// SIMATIC S7-200 project (STEP 7-Micro/WIN), CPU 224 REL 02.00

SYMBOL_TABLE 符号表
AO_B             AQW0     // 板链线变频器DC0-10V信号
AO_X             AQW2     // 悬挂线变频器DC0-10V信号
C_1              C1       // 板链线运行工位计数
C_2              C2       // 悬挂线运行工位计数
HC_0             HC0      // 板链线编码器脉冲检测高速计数器
HC_1             HC1      // 板链线编码器脉冲检测高速计数器
BMQ_B            I0.0     // 板链线编码器
SP_B             I0.1     // 板链线接近开关
SF1_B            I0.2     // 板链线单独启动
SS1_B            I0.3     // 板链线单独停止
SFA_B            I0.4     // 板链线速度微增
SFD_B            I0.5     // 板链线速度微减
BMQ_X            I0.6     // 悬挂线编码器
SP_X             I0.7     // 悬挂线接近开关
SF1_X            I1.0     // 悬挂线单独启动
SS1_X            I1.1     // 悬挂线单独停止
SFA_X            I1.2     // 悬挂线速度微增
SFD_X            I1.3     // 悬挂线速度微减
SF1              I1.4     // 同步连续运行启动
SS1              I1.5     // 同步连续运行停止
BPQ_B            I2.0     // 板链线变频器故障
BPQ_X            I2.1     // 悬挂线变频器故障
SS2              I2.2     // 同步节拍运行停止
SF2              I2.3     // 同步节拍运行启动
M1_0             M1.0     // 板链线单独连续运行
M1_1             M1.1     // 悬挂线单独连续运行
M1_2             M1.2     // 板链线、悬挂线同步节拍运行
M1_3             M1.3     // 板链线、悬挂线同步节拍运行上升沿微分
M1_4             M1.4     // 板链线、悬挂线同步节拍运行状态下板链线接近开关上升沿微分
M1_5             M1.5     // 板链线、悬挂线同步节拍运行状态之板链线运行
M2_4             M2.4     // 板链线、悬挂线同步节拍运行状态下悬挂线接近开关上升沿微分
M2_5             M2.5     // 板链线、悬挂线同步节拍运行状态之悬挂线运行
M2_7             M2.7     // 板链线、悬挂线同步连续运行
M3_0             M3.0     // 板链线变频器复位状态
M3_1             M3.1     // 悬挂线变频器复位状态
M3_4             M3.4     // 单独连续运行开环控制方式
M3_5             M3.5     // 计数器复位
M4_1             M4.1     // C1>C2的下降沿
M4_2             M4.2     // C1<C2的下降沿
HL1              Q0.0     // 同步运行指示
HL2              Q0.1     // 同步停止指示
HL_B             Q0.2     // 板链线单独运行指示
HL_X             Q0.3     // 悬挂线单独运行指示
FWD_B            Q0.4     // 板链线正转
BX1_B            Q0.5     // 板链线自由停止
RST_B            Q0.6     // 板链线变频器复位
FWD_X            Q0.7     // 悬挂线正转
BX1_X            Q1.0     // 悬挂线自由停止
RST_X            Q1.1     // 悬挂线变频器复位
HLA_B            Q2.0     // 板链线速度微增指示
HLD_B            Q2.1     // 板链线速度微减指示
HLA_X            Q2.2     // 悬挂线速度微增指示
HLD_X            Q2.3     // 悬挂线速度微减指示
SM0_0            SM0.0    // 该位始终为1
SM0_1            SM0.1    // 首次扫描时SM0.1=1
SMB_37           SMB37    // HSC0的控制字节
SMB_47           SMB47    // HSC1的控制字节
SMD_38           SMD38    // HSC0的初始值(双整数)
SMD_42           SMD42    // HSC0的预置值(双整数)
SMD_48           SMD48    // HSC1的初始值(双整数)
SMD_52           SMD52    // HSC1的预置值(双整数)
T_0              T0       // 用于检测板链线夹具比悬挂线吊篮早到达接近开关的时间的ms定时器
T_32             T32      // 线体速度计算ms定时器
T_37             T37      // 单独连续运行开环控制状态持续时间
T_40             T40      // 板链线变频器复位持续时间
T_41             T41      // 悬挂线变频器复位持续时间
T_64             T64      // 用于检测悬挂线吊篮比板链线夹具早到达接近开关的时间的ms定时器
T_97             T97      // 板链线频率微增、微减时钟
T_98             T98      // 悬挂线频率微增、微减时钟
T_101            T101     // 板链线、悬挂线同步节拍运行状态下装配（停止）时间
T_105            T105     // 板链线、悬挂线同步连续运行启动时间
T_255            T255     // C1=C2计时
VD_40            VD40     // 板链线设定速度(米/分钟,实数)
VD_60            VD60     // 板链线实际运行速度(米/分钟,实数)
VD_80            VD80     // 悬挂线设定速度(米/分钟,实数)
VD_100           VD100    // 悬挂线实际运行速度(米/分钟,实数)
VD_140           VD140    // 板链线主动链轮节圆周长(米,实数)
VD_160           VD160    // 悬挂线主动链轮节圆周长(米,实数)
VD_240           VD240    // 板链线夹具间距=悬挂线吊篮间距(米,实数)
VD_1800          VD1800   // 线体速度计算采样脉冲数(双整数)
VD_1804          VD1804   // 线体速度计算采样脉冲数(实数)
VD_1854          VD1854   // 检测指定数量脉冲所需要的时间(ms,双整数)
VD_2000          VD2000   // 板链线速度采样周期内的编码器脉冲数(个,双整数)
VD_2004          VD2004   // 板链线速度采样周期内的编码器脉冲数(个,实数)
VD_2008          VD2008   // 板链线编码器的分辨率(个脉冲/转,双整数)
VD_2012          VD2012   // 板链线编码器的分辨率(个脉冲/转,实数)
VD_2016          VD2016   // 线体速度计算采样周期(秒,双整数)
VD_2020          VD2020   // 线体速度计算采样周期(秒,实数)
VD_2024          VD2024   // 板链线速度计算中间值1(实数)
VD_2028          VD2028   // 板链线速度计算中间值2(实数)
VD_2032          VD2032   // 板链线速度计算中间值3(实数)
VD_2100          VD2100   // 检测指定数量脉冲所需要的时间(ms,双整数)
VD_2104          VD2104   // 检测指定数量脉冲所需要的时间(ms,实数)
VD_2108          VD2108   // 悬挂线编码器的分辨率(个脉冲/转,双整数)
VD_2112          VD2112   // 悬挂线编码器的分辨率(个脉冲/转,实数)
VD_2124          VD2124   // 悬挂线速度计算中间值1(实数)
VD_2128          VD2128   // 悬挂线速度计算中间值2(实数)
VD_2132          VD2132   // 悬挂线速度计算中间值3(实数)
VD_2204          VD2204   // 板链线夹具比悬挂线吊篮早到达接近开关的时间(ms,双整数)
VD_2208          VD2208   // 板链线夹具比悬挂线吊篮早到达接近开关的时间(ms,实数)
VD_2212          VD2212   // 速度偏差计算(板链线快)中间变量1
VD_2216          VD2216   // 速度偏差计算(板链线快)中间变量2
VD_2220          VD2220   // 速度偏差计算(板链线快)中间变量3
VD_2224          VD2224   // 速度偏差计算(板链线快)中间变量4
VD_2228          VD2228   // 速度偏差计算(板链线快)中间变量5
VD_2232          VD2232   // 板链线速度-悬挂线速度的值(正值)
VD_2304          VD2304   // 悬挂线吊篮比板链线夹具早到达接近开关的时间(ms,双整数)
VD_2308          VD2308   // 悬挂线吊篮比板链线夹具早到达接近开关的时间(ms,实数)
VD_2312          VD2312   // 速度偏差计算(悬挂线快)中间变量1
VD_2316          VD2316   // 速度偏差计算(悬挂线快)中间变量2
VD_2320          VD2320   // 速度偏差计算(悬挂线快)中间变量3
VD_2324          VD2324   // 速度偏差计算(板链线快)中间变量4
VD_2328          VD2328   // 速度偏差计算(板链线快)中间变量5
VD_2332          VD2332   // 悬挂线速度的值-板链线速度(正值)
VD_2336          VD2336   // 板链线速度-悬挂线速度的值(负值)
VD_2400          VD2400   // 板链线实际运行速度------PID反馈信号处理中间变量1(实数)
VD_2404          VD2404   // 板链线实际运行速度------PID反馈信号处理中间变量2(双整数)
VD_2420          VD2420   // 板链线设定速度------PID设定信号处理结果(实数)
VD_2440          VD2440   // 悬挂线实际运行速度------PID反馈信号处理中间变量1(实数)
VD_2444          VD2444   // 悬挂线实际运行速度------PID反馈信号处理中间变量2(双整数)
VD_2460          VD2460   // 悬挂线单独连续运行、同步节拍运行设定速度------PID设定信号处理中间变量1(实数)
VD_2500          VD2500   // 板链线速度-悬挂线速度的值(实数)
VD_2504          VD2504   // 悬挂线同步连续运行设定速度------PID设定信号处理中间变量2(实数)
VD_2508          VD2508   // 悬挂线同步连续运行设定速度------PID设定信号处理结果
VD_2600          VD2600   // 板链线单独连续开环运行设定速度换算中间变量1(实数)
VD_2604          VD2604   // 板链线单独连续开环运行设定速度换算中间变量2(实数)
VD_2608          VD2608   // 板链线单独连续开环运行设定速度换算中间变量3(双整数)
VD_2700          VD2700   // 悬挂线单独连续开环运行设定速度换算中间变量1(实数)
VD_2704          VD2704   // 悬挂线单独连续开环运行设定速度换算中间变量2(实数)
VD_2708          VD2708   // 悬挂线单独连续开环运行设定速度换算中间变量3(双整数)
VW_122           VW122    // 单独连续运行控制方式（1为开环控制，否则为PID控制）
VW_182           VW182    // 板链线编码器的分辨率(个脉冲/转,整数)
VW_202           VW202    // 悬挂线编码器的分辨率(个脉冲/转,整数)
VW_222           VW222    // 线体速度计算采样脉冲数(整数)
VW_226           VW226    // 线体速度计算采样周期(毫秒,整数)
VW_262           VW262    // PLC复位信号
VW_282           VW282    // 同步节拍运行时间(秒,整数)
VW_1850          VW1850   // 检测指定数量脉冲所需要的时间(ms,整数)
VW_1900          VW1900   // 同步节拍运行时间(百毫秒,整数)
VW_2200          VW2200   // 板链线夹具比悬挂线吊篮早到达接近开关的时间(ms,整数)
VW_2300          VW2300   // 悬挂线吊篮比板链线夹具早到达接近开关的时间(ms,整数)
VW_2408          VW2408   // 板链线实际运行速度------PID反馈信号处理结果(整数)
VW_2448          VW2448   // 悬挂线实际运行速度------PID反馈信号处理结果(整数)
VW_2612          VW2612   // 板链线单独连续开环运行设定速度换算中间变量4(整数)
VW_2712          VW2712   // 悬挂线单独连续开环运行设定速度换算中间变量4(整数)
END_SYMBOL_TABLE

ORGANIZATION_BLOCK 同步控制系统:OB1
TITLE=概要
// 这个PLC程序是给新大洲本田摩托车有限公司上海分公司设计的整车装配板链线和零件输送悬挂线同步控制系统改造工程。
// 项目实现摩托车装配线的自动化生产，通过同步控制板链线和悬挂线的运行来匹配装配节拍。
// 系统支持板链线单独连续运行、悬挂线单独连续运行、同步节拍运行和同步连续运行四种模式，且运行模式互斥。设备要求包含板链线输送设备、悬挂线输送设备、接近开关、高速计数器和变频器。
// 系统启动时，首次扫描标志在 PLC 上电后的第一个周期置 1，触发初始化逻辑。
// 程序支持四种运行模式：板链线单独连续运行、悬挂线单独连续运行、同步节拍运行和同步连续运行，这些模式通过按钮触发，但板链线单独连续运行标志、悬挂线单独连续运行标志、同步节拍运行标志和同步连续运行标志在任意时刻只能有一个为真，其他必须为假，确保车间内不会出现模式冲突导致的生产中断。
BEGIN
Network 1 // 系统初始化
// PLC上电运行的第一个扫描周期执行一次初始化子程序SBR_0，用于程序运行的初始设置
LD     SM0_1:SM0.1
CALL   线体实际速度计算初始化:SBR0
Network 2
// PLC上电运行的第一个扫描周期定义系统参数
LD     SM0_1:SM0.1
MOVR   1.37288, VD_140:VD140
MOVR   0.524271, VD_160:VD160
MOVR   2.4, VD_240:VD240
MOVW   360, VW_182:VW182
MOVW   360, VW_202:VW202
MOVW   50, VW_222:VW222
Network 3 // 板链线单独连续运行
// 板链线单独连续启动、停止、运行指示
LD     SF1_B:I0.2
O      M1_0:M1.0
AN     SS1_B:I0.3
AN     BPQ_B:I2.0
AN     M1_2:M1.2
AN     M2_7:M2.7
=      M1_0:M1.0
=      HL_B:Q0.2
Network 4 // 悬挂线单独连续运行
// 悬挂线单独连续启动、停止、运行指示
LD     SF1_X:I1.0
O      M1_1:M1.1
AN     SS1_X:I1.1
AN     BPQ_X:I2.1
AN     M1_2:M1.2
AN     M2_7:M2.7
=      M1_1:M1.1
=      HL_X:Q0.3
Network 5 // 板链线、悬挂线同步节拍运行
// 板链线、悬挂线同步节拍启动、停止
LD     SF2:I2.3
O      M1_2:M1.2
AN     SS2:I2.2
AN     BPQ_B:I2.0
AN     BPQ_X:I2.1
AN     M1_0:M1.0
AN     M2_7:M2.7
=      M1_2:M1.2
Network 6 // 板链线、悬挂线节拍同步运行装配（停止）时间单位转换
// 把节拍同步运行装配（停止）时间由秒转换为百毫秒
LD     M1_2:M1.2
MOVW   VW_282:VW282, VW_1900:VW1900
*I     +10, VW_1900:VW1900
Network 7 // 板链线、悬挂线同步节拍运行上升沿微分
LD     M1_2:M1.2
EU
=      M1_3:M1.3
Network 8 // 板链线、悬挂线同步节拍运行状态下板链线接近开关上升沿微分
LD     M1_2:M1.2
A      SP_B:I0.1
EU
=      M1_4:M1.4
Network 9 // 板链线、悬挂线同步节拍运行状态之板链线运行
LD     M1_3:M1.3
O      M1_5:M1.5
O      T_101:T101
A      M1_2:M1.2
AN     M1_4:M1.4
=      M1_5:M1.5
Network 10 // 板链线、悬挂线同步节拍运行状态下装配（停止）时间
LD     M1_2:M1.2
AN     M1_5:M1.5
TON    T_101:T101, VW_1900:VW1900
Network 11 // 板链线、悬挂线同步节拍运行状态下悬挂线接近开关上升沿微分
LD     M1_2:M1.2
A      SP_X:I0.7
EU
=      M2_4:M2.4
Network 12 // 板链线、悬挂线同步节拍运行状态之悬挂线运行
LD     M1_3:M1.3
O      M2_5:M2.5
O      T_101:T101
A      M1_2:M1.2
AN     M2_4:M2.4
=      M2_5:M2.5
Network 13 // 板链线、悬挂线同步连续运行
// 板链线、悬挂线同步连续启动、停止
LD     SF1:I1.4
O      M2_7:M2.7
AN     SS1:I1.5
AN     BPQ_B:I2.0
AN     BPQ_X:I2.1
AN     M1_0:M1.0
AN     M1_2:M1.2
=      M2_7:M2.7
TON    T_105:T105, 30
Network 14 // 板链线、悬挂线同步节拍运行、同步连续运行指示
LD     M1_2:M1.2
O      M2_7:M2.7
=      HL1:Q0.0
Network 15 // 板链线、悬挂线同步节拍停止、同步连续停止指示
LDN    M1_2:M1.2
AN     M2_7:M2.7
=      HL2:Q0.1
Network 16 // 板链线变频器运行
LD     M1_0:M1.0
O      M1_5:M1.5
O      T_105:T105
=      FWD_B:Q0.4
Network 17 // 悬挂线变频器运行
LD     M1_1:M1.1
O      M2_5:M2.5
O      T_105:T105
=      FWD_X:Q0.7
Network 18 // 板链线变频器自由停车信号
LD     BPQ_B:I2.0
=      BX1_B:Q0.5
Network 19 // 板链线变频器复位信号（解除变频器报警跳闸状态）
LD     BPQ_B:I2.0
ED
O      M3_0:M3.0
AN     T_40:T40
=      M3_0:M3.0
TON    T_40:T40, 50
=      RST_B:Q0.6
Network 20 // 悬挂线变频器自由停车信号
LD     BPQ_X:I2.1
=      BX1_X:Q1.0
Network 21 // 悬挂线变频器复位信号（解除变频器报警跳闸状态）
LD     BPQ_X:I2.1
ED
O      M3_1:M3.1
AN     T_41:T41
=      M3_1:M3.1
TON    T_41:T41, 50
=      RST_X:Q1.1
Network 22 // 板链线、悬挂线实际运行速度检测
LD     SM0_0:SM0.0
CALL   线体实际运行速度检测:SBR1
Network 23 // 板链线实际运行速度计算
LD     SM0_0:SM0.0
CALL   板链线实际运行速度计算:SBR2
Network 24 // 悬挂线实际运行速度计算
LD     SM0_0:SM0.0
CALL   悬挂线实际运行速度计算:SBR3
Network 25 // 线体实际速度偏差检测
LD     M2_7:M2.7
CALL   线体实际速度偏差检测:SBR4
Network 26 // 速度偏差计算_板链线快
LD     M4_1:M4.1
CALL   速度偏差计算_板链线快:SBR5
Network 27 // 速度偏差计算_悬挂线快
LD     M4_2:M4.2
CALL   速度偏差计算_悬挂线快:SBR6
Network 28 // PID设定及反馈信号处理
LD     SM0_0:SM0.0
CALL   PID设定及反馈信号处理:SBR13
Network 29 // 板链线、悬挂线单独运行开环控制检测
LDW=   VW_122:VW122, 1
=      M3_4:M3.4
TON    T_37:T37, 10
Network 30 // 板链线单独连续运行开环控制
LD     M1_0:M1.0
A      T_37:T37
CALL   板链线单独连续开环运行:SBR14
Network 31
LD     M1_0:M1.0
AN     T_37:T37
=      M10.1
Network 32 // 板链线单独连续运行PID控制（转换为手动时实现无扰切换------不会存在PID输出值为0输出的扫描周期，在该工程中没有实际意义，这里只是提出了一个编程思想）
LD     SM0_0:SM0.0
CALL   PID0_INIT:SBR7, VW_2408:VW2408, VD_2420:VD2420, M10.1, 0.3, VW5000
Network 33
LD     M1_0:M1.0
AN     T_37:T37
MOVW   VW5000, AO_B:AQW0
Network 34 // 悬挂线单独连续运行开环控制
LD     M1_1:M1.1
A      T_37:T37
CALL   悬挂线单独连续开环运行:SBR15
Network 35
LD     M1_1:M1.1
AN     T_37:T37
=      M10.2
Network 36 // 悬挂线单独连续运行PID控制（转换为手动时实现无扰切换------不会存在PID输出值为0输出的扫描周期，在该工程中没有实际意义，这里只是提出了一个编程思想）
LD     SM0_0:SM0.0
CALL   PID1_INIT:SBR8, VW_2448:VW2448, VD_2460:VD2460, M10.2, 0.3, VW5100
Network 37
LD     M1_1:M1.1
AN     T_37:T37
MOVW   VW5100, AO_X:AQW2
Network 38
LD     SM0_0:SM0.0
CALL   PID2_INIT:SBR9, VW_2408:VW2408, VD_2420:VD2420, M1_2:M1.2, 0.3, VW5004
Network 39 // 板链线、悬挂线同步节拍运行PID控制
LD     SM0_0:SM0.0
CALL   PID3_INIT:SBR10, VW_2448:VW2448, VD_2460:VD2460, M1_2:M1.2, 0.3, VW5104
Network 40
LD     M1_2:M1.2
MOVW   VW5004, AO_B:AQW0
MOVW   VW5104, AO_X:AQW2
Network 41
LD     SM0_0:SM0.0
CALL   PID4_INIT:SBR11, VW_2408:VW2408, VD_2420:VD2420, M2_7:M2.7, 0.3, VW5008
Network 42
LD     SM0_0:SM0.0
CALL   PID5_INIT:SBR12, VW_2448:VW2448, VD_2508:VD2508, M2_7:M2.7, 0.3, VW5108
Network 43
LD     M2_7:M2.7
MOVW   VW5008, AO_B:AQW0
MOVW   VW5108, AO_X:AQW2
Network 44 // 使能TD200文本显示器消息
LD     SM0_0:SM0.0
=      V14.7
=      V14.6
=      V14.5
=      V14.4
=      V14.2
=      V14.1
=      V14.0
=      V15.7
=      V15.6
=      V15.5
=      V15.2
=      V15.1
=      V15.0
END_ORGANIZATION_BLOCK

SUBROUTINE_BLOCK 线体实际速度计算初始化:SBR0
TITLE=初始化子程序，主要完成系统初始化，对各内部变量、中间变量进行置位或复位
BEGIN
Network 1 // HSC0初始化子程序
// 设置HSC0控制字节SMB37的值为16进制数据F8（赋值为16#F8，也可以用二进制表示（赋值2#11111000））：SM37.0=0高电平复位，SM37.1=0（系统保留），SM37.2=0正交计数器四倍速方式（当计数器模式设为9~11时才有用），SM37.3=1增计数，SM37.4=1更新方向，SM37.5=1向HSC0写入新的预置值，SM37.6=1向HSC0写入新的初始值，SM37.7=1高速计数器HSC0有效；
// 设置高速计数器HC0工作模式为0：带有内部方向控制的单相计数器，输入点为I0.0；
// 将HSC0的初始值寄存器SMD38的值设置为0；
// 执行HSC指令，将控制字节SMB37、初始值/预置值寄存器（SMD38/SMD42）以及工作模式写入高速计数器HSC0；
LD     SM0_1:SM0.1
MOVB   16#F8, SMB_37:SMB37
HDEF   0, 0
MOVD   +0, SMD_38:SMD38
MOVD   VD_1800:VD1800, SMD_42:SMD42
ATCH   高速计数器0中断:INT1, 12
ENI
HSC    0
Network 2 // HSC1初始化子程序
// 程序注释与"HSC0初始化"子程序注释类同，此处不再赘述。
LD     SM0_1:SM0.1
MOVB   16#F8, SMB_47:SMB47
HDEF   1, 0
MOVD   +0, SMD_48:SMD48
MOVD   VD_1800:VD1800, SMD_52:SMD52
ATCH   高速计数器1中断:INT2, 13
ENI
HSC    1
END_SUBROUTINE_BLOCK

SUBROUTINE_BLOCK 线体实际运行速度检测:SBR1
TITLE=板链线、悬挂线实际运行速度检测
BEGIN
Network 1
LDD>   HC_0:HC0, VD3000
MOVD   +0, SMD_38:SMD38
MOVD   VD3000, SMD_42:SMD42
MOVB   16#F8, SMB_37:SMB37
HSC    0
Network 2
LDD>   HC_1:HC1, VD_1800:VD1800
MOVD   +0, SMD_48:SMD48
MOVD   VD_1800:VD1800, SMD_52:SMD52
MOVB   16#F8, SMB_47:SMB47
HSC    1
END_SUBROUTINE_BLOCK

SUBROUTINE_BLOCK 板链线实际运行速度计算:SBR2
TITLE=板链线实际运行速度计算
BEGIN
Network 1
LD     M1_0:M1.0
O      M1_2:M1.2
O      M2_7:M2.7
ITD    VW_222:VW222, VD3000
Network 2
LDN    M1_0:M1.0
AN     M1_2:M1.2
AN     M2_7:M2.7
MOVR   0.0, VD_60:VD60
Network 3
// 当线体运行速度检测采样时钟脉冲到来时进行以下动作：
// 将高速计数器HSC0的当前值HC0（在采样周期内测得的编码器脉冲数）传送到VD存储器；
// 将HSC0的初始值寄存器SMD38的值设置为0，为下一个线体速度检测采样周期做准备；
// 设置HSC0控制字节SMB37的值为16进制数据F8（赋值为16#F8，也可以用二进制表示（赋值2#11111000））：SM37.0=0高电平复位，SM37.1=0（系统保留），SM37.2=0正交计数器四倍速方式（当计数器模式设为9~11时才有用），SM37.3=1增计数，SM37.4=1更新方向，SM37.5=1向HSC0写入新的预置值，SM37.6=1向HSC0写入新的初始值，SM37.7=1高速计数器HSC0有效；为下一个线体速度检测采样周期做准备；
// 将板链线速度采样周期内的编码器脉冲数（个，双整数）转换为板链线速度采样周期内的编码器脉冲数（个，实数）；
// 将编码器的分辨率（个脉冲/转，整数）转换为编码器的分辨率（个脉冲/转，双整数）；
// 将编码器的分辨率（个脉冲/转，双整数）转换为编码器的分辨率（个脉冲/转，实整数）；
// 将线体速度计算采样周期（秒，整数）转换为线体速度计算采样周期（秒，双整数）；
// 将线体速度计算采样周期（秒，双整数）转换为线体速度计算采样周期（秒，实数）；
// 然后根据在线体速度计算采样周期T（单位：秒）、在采样周期内测得的编码器脉冲数M、编码器的分辨率P（编码器每转一圈产生的脉冲数）、线体主动链轮节圆的周长L（单位：米）来计算：V（米/分钟）=（60 × M  × L）÷（P × T）：
// 计算【板链线速度采样周期内的编码器脉冲数 × 板链线主动链轮节圆周长】的值；
// 计算【板链线速度采样周期内的编码器脉冲数 × 板链线主动链轮节圆周长 × 60】的值；
// 计算【板链线速度采样周期内的编码器脉冲数 × 板链线主动链轮节圆周长 × 60 ÷ 编码器的分辨率】的值；
// 计算【板链线速度采样周期内的编码器脉冲数 × 板链线主动链轮节圆周长 × 60 ÷ 编码器的分辨率 ÷ 线体速度计算采样周期】的值，这个值就是板链线的实际运行速度。
LD     M1_0:M1.0
O      M1_2:M1.2
O      M2_7:M2.7
ITD    VW1950, VD1954
MOVD   VD1954, VD_2000:VD2000
DTR    VD_2000:VD2000, VD_2004:VD2004
ITD    VW_182:VW182, VD_2008:VD2008
DTR    VD_2008:VD2008, VD_2012:VD2012
DTR    VD3000, VD1824
MOVR   VD1824, VD_2024:VD2024
*R     VD_140:VD140, VD_2024:VD2024
MOVR   VD_2024:VD2024, VD_2028:VD2028
*R     60000.0, VD_2028:VD2028
MOVR   VD_2028:VD2028, VD_2032:VD2032
/R     VD_2012:VD2012, VD_2032:VD2032
AR<>   VD_2004:VD2004, 0.0
AR<    VD_2004:VD2004, 32760.0
MOVR   VD_2032:VD2032, VD_60:VD60
/R     VD_2004:VD2004, VD_60:VD60
END_SUBROUTINE_BLOCK

SUBROUTINE_BLOCK 悬挂线实际运行速度计算:SBR3
TITLE=悬挂线实际运行速度计算
BEGIN
Network 1
LD     M1_1:M1.1
O      M1_2:M1.2
O      M2_7:M2.7
ITD    VW_222:VW222, VD_1800:VD1800
Network 2
LDN    M1_1:M1.1
AN     M1_2:M1.2
AN     M2_7:M2.7
MOVR   0.0, VD_100:VD100
Network 3
// 程序注释与"板链线实际运行速度计算"子程序注释类同，此处不再赘述。
LD     M1_1:M1.1
O      M1_2:M1.2
O      M2_7:M2.7
ITD    VW_1850:VW1850, VD_1854:VD1854
MOVD   VD_1854:VD1854, VD_2100:VD2100
DTR    VD_2100:VD2100, VD_2104:VD2104
ITD    VW_202:VW202, VD_2108:VD2108
DTR    VD_2108:VD2108, VD_2112:VD2112
DTR    VD_1800:VD1800, VD_1804:VD1804
MOVR   VD_1804:VD1804, VD_2124:VD2124
*R     VD_160:VD160, VD_2124:VD2124
MOVR   VD_2124:VD2124, VD_2128:VD2128
*R     60000.0, VD_2128:VD2128
MOVR   VD_2128:VD2128, VD_2132:VD2132
/R     VD_2112:VD2112, VD_2132:VD2132
AR<>   VD_2104:VD2104, 0.0
AR<    VD_2104:VD2104, 32760.0
MOVR   VD_2132:VD2132, VD_100:VD100
/R     VD_2104:VD2104, VD_100:VD100
END_SUBROUTINE_BLOCK

SUBROUTINE_BLOCK 线体实际速度偏差检测:SBR4
TITLE=板链线、悬挂线实际运行速度偏差检测
BEGIN
Network 1 // 对板链线运行的工位数进行计数
LD     M2_7:M2.7
A      SP_B:I0.1
LD     M3_5:M3.5
CTU    C_1:C1, 32767
Network 2 // 对悬挂线运行的工位数进行计数
LD     M2_7:M2.7
A      SP_X:I0.7
LD     M3_5:M3.5
CTU    C_2:C2, 32767
Network 3 // 计数器复位
LDW=   C_1:C1, C_2:C2
AW>=   C_1:C1, 30000
OW=    VW_262:VW262, 1
OW>=   T_0:T0, 20000
OW>=   T_64:T64, 20000
=      M3_5:M3.5
Network 4
LDW>=  T_0:T0, 20000
MOVW   0, T_0:T0
Network 5
LDW>=  T_64:T64, 20000
MOVW   0, T_64:T64
Network 6 // 检测板链线夹具比悬挂线吊篮早到达接近开关的时间
LDW>   C_1:C1, C_2:C2
TONR   T_0:T0, 32767
Network 7 // 板链线夹具到达板链线接近开关后，悬挂线吊篮到达悬挂线接近开关的时间点
LDW>   C_1:C1, C_2:C2
ED
=      M4_1:M4.1
Network 8 // 检测悬挂线吊篮比板链线夹具早到达接近开关的时间
LDW<   C_1:C1, C_2:C2
TONR   T_64:T64, 32767
Network 9 // 悬挂线吊篮到达悬挂线接近开关后，板链线夹具到达板链线接近开关的时间点
LDW<   C_1:C1, C_2:C2
ED
=      M4_2:M4.2
Network 10 // C1=C2计时
LDW=   C_1:C1, C_2:C2
TON    T_255:T255, 10
Network 11 // 线体实际运行偏差时间清零
LD     T_255:T255
MOVW   0, T_0:T0
MOVW   0, T_64:T64
END_SUBROUTINE_BLOCK

SUBROUTINE_BLOCK 速度偏差计算_板链线快:SBR5
TITLE=速度偏差计算_板链线快
BEGIN
Network 1 // 计算板链线速度-悬挂线速度的值（正值）
// 在板链线夹具到达板链线接近开关后，当悬挂线吊篮到达悬挂线接近开关时，计算板链线速度-悬挂线速度的值。具体控制算法请参阅控制方案，此处不再赘述。
// 将检测板链线夹具比悬挂线吊篮早到达接近开关的时间传送到变量VW2200（整数）；
// 将变量VW2200（整数）转换为变量VD2204（双整数）；
// 将变量VW2204（双整数）转换为变量VD2208（实数）；
// 将变量VD2208（实数）乘以板链线实际运行速度VD60（米/分钟，实数）得到变量VD2212（实数）；
// 将变量VD2212（实数）乘以板链线实际运行速度VD60（米/分钟，实数）得到变量VD2216（实数）；
// 将变量VD240（实数）乘以60000.0（实数）得到变量VD2220（实数）；
// 将板链线实际运行速度VD60（米/分钟，实数）乘以变量VD2208（实数）得到变量VD2224（实数）；
// 将变量VD2220（实数）加上变量VD2224（实数）得到变量VD2228（实数）；
// 将变量VD2228（实数）除以变量VD2228（实数）得到变量VD2232（实数）；
// 将变量VD2232（板链线速度-悬挂线速度的值（正值），实数）传送到变量VD2500。
LD     M4_1:M4.1
LPS
MOVW   T_0:T0, VW_2200:VW2200
ITD    VW_2200:VW2200, VD_2204:VD2204
DTR    VD_2204:VD2204, VD_2208:VD2208
MOVR   VD_2208:VD2208, VD_2212:VD2212
*R     VD_60:VD60, VD_2212:VD2212
MOVR   VD_2212:VD2212, VD_2216:VD2216
*R     VD_60:VD60, VD_2216:VD2216
MOVR   VD_240:VD240, VD_2220:VD2220
*R     60000.0, VD_2220:VD2220
MOVR   VD_60:VD60, VD_2224:VD2224
*R     VD_2208:VD2208, VD_2224:VD2224
MOVR   VD_2220:VD2220, VD_2228:VD2228
+R     VD_2224:VD2224, VD_2228:VD2228
AR<>   VD_2228:VD2228, 0.0
MOVR   VD_2216:VD2216, VD_2232:VD2232
/R     VD_2228:VD2228, VD_2232:VD2232
LPP
MOVR   VD_2232:VD2232, VD_2500:VD2500
END_SUBROUTINE_BLOCK

SUBROUTINE_BLOCK 速度偏差计算_悬挂线快:SBR6
TITLE=速度偏差计算_悬挂线快
BEGIN
Network 1 // 计算板链线速度-悬挂线速度的值（负值）
// 程序注释与"速度偏差计算_板链线快"子程序注释类同，此处不再赘述。
LD     M4_2:M4.2
MOVW   T_64:T64, VW_2300:VW2300
ITD    VW_2300:VW2300, VD_2304:VD2304
DTR    VD_2304:VD2304, VD_2308:VD2308
MOVR   VD_2308:VD2308, VD_2312:VD2312
*R     VD_60:VD60, VD_2312:VD2312
MOVR   VD_2312:VD2312, VD_2316:VD2316
*R     VD_60:VD60, VD_2316:VD2316
MOVR   VD_240:VD240, VD_2320:VD2320
*R     60000.0, VD_2320:VD2320
MOVR   VD_60:VD60, VD_2324:VD2324
*R     VD_2308:VD2308, VD_2324:VD2324
MOVR   VD_2320:VD2320, VD_2328:VD2328
-R     VD_2324:VD2324, VD_2328:VD2328
MOVR   VD_2316:VD2316, VD_2332:VD2332
/R     VD_2328:VD2328, VD_2332:VD2332
MOVR   VD_2332:VD2332, VD_2336:VD2336
/R     -1.0, VD_2336:VD2336
MOVR   VD_2336:VD2336, VD_2500:VD2500
END_SUBROUTINE_BLOCK

// SBR7: protected block, not included

// SBR8: protected block, not included

// SBR9: protected block, not included

// SBR10: protected block, not included

// SBR11: protected block, not included

// SBR12: protected block, not included

SUBROUTINE_BLOCK PID设定及反馈信号处理:SBR13
TITLE=PID设定信号、反馈信号处理
BEGIN
Network 1 // 板链线实际运行速度------PID反馈信号处理
// PID反馈信号处理：因为设定速度在0.0~10.0米/分钟之间，而PID控制器的设定值是整数而不是实数，采用取整或四舍五入的方式都无法保证控制的精确性，所以考虑将设定值乘以1000.0以后再取整并转化为实数，将信号放大并处理后后送至PID控制器，控制精确度就比较高了。当然，既然设定速度乘以了1000，那么反馈值也得乘以1000。
// 将板链线实际运行速度（米/分钟，实数）乘以1000.0得到变量VD2400（实数）；
// 将变量VD2400（实数）取整得到变量VD2404（双整数）；
// 将变量VD2404（双整数）转换为变量VW2408（整数）------PID控制器只接受整数类型的反馈值。
LD     SM0_0:SM0.0
MOVR   VD_60:VD60, VD_2400:VD2400
*R     1000.0, VD_2400:VD2400
ROUND  VD_2400:VD2400, VD_2404:VD2404
DTI    VD_2404:VD2404, VW_2408:VW2408
Network 2 // 板链线设定速度------PID设定信号处理
// 将板链线设定速度（米/分钟，实数）乘以1000.0得到变量VD2420（实数）；
LD     SM0_0:SM0.0
MOVR   VD_40:VD40, VD_2420:VD2420
*R     1000.0, VD_2420:VD2420
Network 3 // 悬挂线实际运行速度------PID反馈信号处理
// 程序注释与"板链线实际运行速度------PID反馈信号处理"程序段注释类同，此处不再赘述。
LD     SM0_0:SM0.0
MOVR   VD_100:VD100, VD_2440:VD2440
*R     1000.0, VD_2440:VD2440
ROUND  VD_2440:VD2440, VD_2444:VD2444
DTI    VD_2444:VD2444, VW_2448:VW2448
Network 4 // 悬挂线单独连续运行、同步节拍运行设定速度------PID设定信号处理
// 将悬挂线设定速度（米/分钟，实数）乘以1000.0得到变量VD2460（实数）；
LD     SM0_0:SM0.0
MOVR   VD_80:VD80, VD_2460:VD2460
*R     1000.0, VD_2460:VD2460
Network 5 // 悬挂线同步连续运行设定速度------PID设定信号处理
// 将板链线速度---悬挂线速度的值（实数）乘以1000.0得到变量VD2504（实数）；
// 将变量VD2460（实数）加上变量VD2504（实数）得到变量VD2508（实数）。
LD     SM0_0:SM0.0
MOVR   VD_2500:VD2500, VD_2504:VD2504
*R     1000.0, VD_2504:VD2504
MOVR   VD_2460:VD2460, VD_2508:VD2508
+R     VD_2504:VD2504, VD_2508:VD2508
END_SUBROUTINE_BLOCK

SUBROUTINE_BLOCK 板链线单独连续开环运行:SBR14
TITLE=板链线单独连续开环运行
BEGIN
Network 1 // 设定速度换算
LD     M1_0:M1.0
A      T_37:T37
MOVR   VD_40:VD40, VD_2600:VD2600
*R     1.333, VD_2600:VD2600
MOVR   VD_2600:VD2600, VD_2604:VD2604
*R     3200.0, VD_2604:VD2604
ROUND  VD_2604:VD2604, VD_2608:VD2608
DTI    VD_2608:VD2608, VW_2612:VW2612
MOVW   VW_2612:VW2612, AO_B:AQW0
Network 2 // 板链线频率微增、微减时钟设置
LD     M1_0:M1.0
A      T_37:T37
AN     T_97:T97
TON    T_97:T97, 5
Network 3 // 频率微增
LD     M1_0:M1.0
A      T_37:T37
A      T_97:T97
A      SFA_B:I0.4
AN     SFD_B:I0.5
+R     0.001, VD_40:VD40
Network 4 // 频率微减
LD     M1_0:M1.0
A      T_37:T37
A      T_97:T97
A      SFD_B:I0.5
AN     SFA_B:I0.4
-R     0.001, VD_40:VD40
Network 5 // 频率微增、微减指示
LD     M1_0:M1.0
A      T_37:T37
LPS
A      SFA_B:I0.4
AN     SFD_B:I0.5
=      HLA_B:Q2.0
LPP
A      SFD_B:I0.5
AN     SFA_B:I0.4
=      HLD_B:Q2.1
END_SUBROUTINE_BLOCK

SUBROUTINE_BLOCK 悬挂线单独连续开环运行:SBR15
TITLE=悬挂线单独连续开环运行
BEGIN
Network 1
LD     M1_1:M1.1
A      T_37:T37
MOVR   VD_80:VD80, VD_2700:VD2700
*R     1.333, VD_2700:VD2700
MOVR   VD_2700:VD2700, VD_2704:VD2704
*R     3200.0, VD_2704:VD2704
ROUND  VD_2704:VD2704, VD_2708:VD2708
DTI    VD_2708:VD2708, VW_2712:VW2712
MOVW   VW_2712:VW2712, AO_X:AQW2
Network 2 // 悬挂线频率微增、微减时钟设置
LD     M1_1:M1.1
A      T_37:T37
AN     T_98:T98
TON    T_98:T98, 5
Network 3 // 频率微增
LD     M1_1:M1.1
A      T_37:T37
A      T_98:T98
A      SFA_X:I1.2
AN     SFD_X:I1.3
+R     0.001, VD_80:VD80
Network 4 // 频率微减
LD     M1_1:M1.1
A      T_37:T37
A      T_98:T98
A      SFD_X:I1.3
AN     SFA_X:I1.2
-R     0.001, VD_80:VD80
Network 5 // 频率微增、微减指示
LD     M1_1:M1.1
A      T_37:T37
LPS
A      SFA_X:I1.2
AN     SFD_X:I1.3
=      HLA_X:Q2.2
LPP
A      SFD_X:I1.3
AN     SFA_X:I1.2
=      HLD_X:Q2.3
END_SUBROUTINE_BLOCK

// INT0: protected block, not included

INTERRUPT_BLOCK 高速计数器0中断:INT1
TITLE=中断程序注释
BEGIN
Network 1 // 网络标题
// 网络注释
LD     SM0_0:SM0.0
MOVW   T96, VW1950
Network 2
LDN    SM0_0:SM0.0
TON    T96, 32767
Network 3
LD     SM0_0:SM0.0
MOVD   +0, SMD_38:SMD38
MOVD   VD3000, SMD_42:SMD42
MOVB   16#F8, SMB_37:SMB37
HSC    0
TON    T96, 32767
END_INTERRUPT_BLOCK

INTERRUPT_BLOCK 高速计数器1中断:INT2
TITLE=中断程序注释
BEGIN
Network 1
LD     SM0_0:SM0.0
MOVW   T_32:T32, VW_1850:VW1850
Network 2
LDN    SM0_0:SM0.0
TON    T_32:T32, 32767
Network 3 // 网络标题
// 网络注释
LD     SM0_0:SM0.0
MOVD   +0, SMD_48:SMD48
MOVD   VD_1800:VD1800, SMD_52:SMD52
MOVB   16#F8, SMB_47:SMB47
HSC    1
TON    T_32:T32, 32767
END_INTERRUPT_BLOCK

// (further data pages could not be read)
